(* CoDeSys 2.3.9.62 project: Cap6_ej2.pro *)
(* Libraries: Standard.lib 4.10.05 12:14:46, IecSfc.lib*2.6.14 10:37:46 *)

(* POU PLC_PRG, LD *)
PROGRAM PLC_PRG
VAR
    (* Entradas *)
	A: BOOL;
       B:BOOL;
    (* Salidas *)
   	S1: BOOL;
      S2 :BOOL;
    (* Instancias de bloques funcionales *)
	DetectorSubida: R_TRIG;
END_VAR
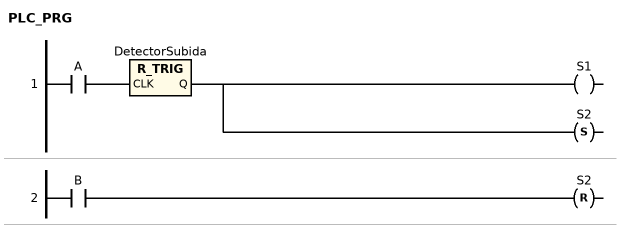
_LD_ (* Ladder Diagram *)
NETWORK 1
	[A] - DetectorSubida:R_TRIG(CLK: *) --- (S1) (S S2)
NETWORK 2
	[B] --- (R S2)
_END_LD_
(* the same logic as Structured Text *)
(* Network 1 *)
DetectorSubida(CLK := A);
S1 := DetectorSubida.Q;
IF DetectorSubida.Q THEN S2 := TRUE; END_IF;
(* Network 2 *)
IF B THEN S2 := FALSE; END_IF;
END_PROGRAM

(* Visualisation Visu
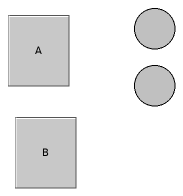
button at (42,51)-(103,122): text "A"; taps PLC_PRG.A
ellipse at (168,44)-(209,85): alarm colour if PLC_PRG.S1
ellipse at (168,101)-(209,142): alarm colour if PLC_PRG.S2
button at (49,153)-(110,224): text "B"; taps PLC_PRG.B
2 elements of other kinds (tables, trends, ...) not read
*)
